{attribute 'qualified_only'} VAR_GLOBAL CONSTANT sDefaultOrg             : STRING(80) := 'ElektroBeckhoff'; sDefaultBucket          : STRING(80) := 'Telemetry'; cnMaxBatchSize          : UDINT      := 500; cnMaxRetries            : UINT       := 3; tDefaultFlushInterval   : TIME       := T#5S; tDefaultRequestTimeout  : TIME       := T#10S; END_VAR

(* stored: Version 1.1.0.1, ProductVersion 3.1.4024.16
   GVL GVL_Sample_ParamInflux: Id {0f17b9d8-2670-4e5d-b543-a16dd48c7f87} *)
